INTERFACE I_PropertyCollection

METHOD PUBLIC GetEnumerator : I_ForwardEnumerator
VAR_INPUT
END_VAR
END_METHOD

METHOD PUBLIC TryGetByName : BOOL
VAR_INPUT
	Name : STRING;
	Destination : REFERENCE TO I_Property;
END_VAR
END_METHOD

END_INTERFACE

(* stored: Version 1.1.0.1, ProductVersion 3.1.4024.12
   Itf I_PropertyCollection: Id {4ba627a9-63df-0edd-30dd-699f1a143552}
   Method GetEnumerator: Id {646f5606-1ba6-07b7-10cd-b19e40dedbba}
   Method TryGetByName: Id {816cfa84-ac0c-0a44-34ec-af16a76d05fb} *)
